Yaskawa INFORM job: SPINDLE_AIR.JBI

/JOB
//NAME SPINDLE_AIR
//POS
///NPOS 0,0,0,0,0,0
//INST
///DATE 2022/03/01 16:21
///ATTR SC,RW
///GROUP1 RB1
NOP
DOUT OT#(17) ON
END
